PROGRAM MAIN
VAR
	fbFIFOTest : FB_FIFOTest;
END_VAR

fbFIFOTest();

END_PROGRAM

(* stored: Version 1.1.0.1, ProductVersion 3.1.4024.2
   POU MAIN: Id {c51feae6-2cfd-4c89-b598-db2fc7fdb705}, SpecialFunc None *)
